// TIA Portal V17 export
// export: Created 2022-07-28T18:02:44.8373404Z, ExportSetting None, DisplayName Totally Integrated Automation Portal, DisplayVersion V17, DisplayName TIA Portal Openness, DisplayVersion V17, DisplayName TIA Portal Teamcenter Gateway, DisplayVersion V17, DisplayName TIA Portal Version Control Interface, DisplayVersion V17, DisplayName TIA Portal Test Suite Advanced, DisplayVersion V17, DisplayName SINAMICS Startdrive Advanced, DisplayVersion V17, DisplayName SINAMICS DCC, DisplayVersion V17, DisplayName SINAMICS Startdrive G130, G150, S120, S150, SINAMICS MV, S210, DisplayVersion V17, DisplayName SINAMICS Startdrive G110M, G120, G120C, G120D, G120P, G115D, DisplayVersion V17, DisplayName STEP 7 Professional, DisplayVersion V17, DisplayName SIMATIC Energy Suite, DisplayVersion V17, DisplayName STEP 7 CFC, DisplayVersion V17, DisplayName STEP 7 Safety, DisplayVersion V17, DisplayName WinCC Advanced / Unified PC, DisplayVersion V17, DisplayName SIMATIC Visualization Architect, DisplayVersion V17
FUNCTION_BLOCK "Lib_FB_PLC"   // FB1, SCL
{ S7_Optimized_Access := 'TRUE' }
// stored: MemoryReserve 500, SetENOAutomatically false
   VAR_IN_OUT
      IO_PLC : "Lib_UDT_PLC";
   END_VAR
   VAR
      TMBITS_PREV : Int;   // попереднє значення таймерних меандрів
      MEM_RUNTIME : LReal;   // память для вимірювання часу циклу
      FB_LTIME : LReal;
      FB_LTIME_1 : Real;
      TIME_TCK_ms : LReal;
      TIME_TCK_s : LReal;
      TIME_TCK_min : Real;
      TIME_TCK_ms_1 : DInt;
      TIME_TCK_ms_2 : UDInt;
      TIME_TCK_ms_3 : DInt;
      TIME_TCK_min_3rs : Real;
      OB1 : Struct
         PrevOutputTime : Date_And_Time;   // Время на предыдущего вызова
         cyclicTime : Int;   // Время цыкла (мс)
      END_STRUCT;
      TIME_ZONE : Struct
         Set : Bool;
         DONE : Bool;
         BUSY : Bool;
         ERROR : Bool;
         STATUS : Word;
         TimeTransformationRule : TimeTransformationRule;
      END_STRUCT;
      SET_TIMEZONE_Instance { ExternalAccessible := 'False'; ExternalVisible := 'False'; ExternalWritable := 'False'} : SET_TIMEZONE;
   END_VAR
   VAR_TEMP
      TMBITS_CUR : Int;
      RESULT : Int;
      i : Int;
      NOW : DTL;
      retVal : Int;
      test : LReal;
      TaskTimeMax : LTime;
      TaskTimeMin : LTime;
      TaskTimeLive : LTime;
      returnValue : Int;
   END_VAR
   // TIME_ZONE.TimeTransformationRule.Bias := 120;
   // TIME_ZONE.TimeTransformationRule.DaylightBias := 60;
   // TIME_ZONE.TimeTransformationRule.DaylightStartMonth := 3;
   // TIME_ZONE.TimeTransformationRule.DaylightStartWeek := 5;
   // TIME_ZONE.TimeTransformationRule.DaylightStartWeekday := 1;
   // TIME_ZONE.TimeTransformationRule.DaylightStartHour := 3;
   // TIME_ZONE.TimeTransformationRule.DaylightStartMinute := 0;
   // TIME_ZONE.TimeTransformationRule.StandardStartMonth := 10;
   // TIME_ZONE.TimeTransformationRule.StandardStartWeek := 5;
   // TIME_ZONE.TimeTransformationRule.StandardStartWeekday := 1;
   // TIME_ZONE.TimeTransformationRule.StandardStartHour := 3;
   // TIME_ZONE.TimeTransformationRule.StandardStartMinute := 0;
   // TIME_ZONE.TimeTransformationRule.TimeZoneName := '(GMT+02:00) Helsinki, Kiev, Riga, Sofia, Tallinn, Vilnius';
BEGIN
   //#FB_LTIME := RUNTIME(#MEM_RUNTIME) * 1000.0;



       REGION Iніціалізація "FirstScan"
           #IO_PLC.PLS.FirstScan := "FirstScan";
           IF #IO_PLC.PLS.FirstScan THEN (*при першому скані*)
               #IO_PLC.ID := 1;             (*Ідентифікатор завжди 1*)
               #IO_PLC.TIME_TCK.Time1cycle_r := 0;
               #TMBITS_CUR := 0;
               #TMBITS_PREV := 0;
           END_IF;
       END_REGION



   REGION таймерні біти та лічильники
       (*плинні значення*)
       REGION плинні значення
           #TMBITS_CUR.%X0 := "Clock_10Hz";         // 100MS 
           #TMBITS_CUR.%X1 := "Clock_5Hz";        // 200MS
           #TMBITS_CUR.%X2 := "Clock_2Hz";        // 500MS
           #TMBITS_CUR.%X3 := "Clock_1Hz";      // 1S
           #TMBITS_CUR.%X7 := #IO_PLC.NOW[0] > 16#29; //min
       END_REGION
       (*відловлювання імпульсів необхідних часових періодів*)
       REGION відловлювання імпульсів необхідних часових періодів
           #IO_PLC.PLS.P100MS := #TMBITS_CUR.%X0 AND NOT #TMBITS_PREV.%X0; (*100 мс *)
           #IO_PLC.PLS.P200MS := #TMBITS_CUR.%X1 AND NOT #TMBITS_PREV.%X1; (*200 мс*)
           #IO_PLC.PLS.P500MS := #TMBITS_CUR.%X2 AND NOT #TMBITS_PREV.%X2; (*500 мс*)
           #IO_PLC.PLS.P1S := #TMBITS_CUR.%X3 AND NOT #TMBITS_PREV.%X3; (*1 с*)
           #IO_PLC.PLS.P60S := #TMBITS_CUR.%X7 AND NOT #TMBITS_PREV.%X7; (*1 хв*)
       END_REGION
       (*підрахунок кількості секунд і хвилин*)
       (*загальний час з початку 1-го циклу контролера (в секундах)*)
       REGION загальний час з початку 1-го циклу контролера (в секундах)
           IF #IO_PLC.PLS.P1S THEN
               #IO_PLC.TIME_TCK.Time1cycle_di := #IO_PLC.TIME_TCK.Time1cycle_di + 1;
           END_IF;
           IF #IO_PLC.TIME_TCK.Time1cycle_di > 16#7FFF_FFFF THEN
               #IO_PLC.TIME_TCK.Time1cycle_di := 16#7FFF_FFFF;
           END_IF;
       END_REGION
       (*загальний час роботи ПЛК з моменту пуску (в хвилинах)*)
       REGION загальний час роботи ПЛК з моменту пуску (в хвилинах)
           IF #IO_PLC.PLS.P60S AND NOT #IO_PLC.PLS.FirstScan THEN
               #IO_PLC.TIME_TCK.TimeTotalPLC := #IO_PLC.TIME_TCK.TimeTotalPLC + 1;
           END_IF;
           IF #IO_PLC.TIME_TCK.TimeTotalPLC > 16#7FFF_FFFF THEN
               #IO_PLC.TIME_TCK.TimeTotalPLC := 16#7FFF_FFFF;
           END_IF;
       END_REGION
       (*розрахунок інших часових періодів*)
       REGION розрахунок інших часових періодів
           #IO_PLC.PLS.P2S := (#IO_PLC.TIME_TCK.Time1cycle_di MOD 2) = 0 AND #IO_PLC.PLS.P1S;(*2 с*)
           #IO_PLC.PLS.P5S := (#IO_PLC.TIME_TCK.Time1cycle_di MOD 5) = 0 AND #IO_PLC.PLS.P1S;(*5 с*)
           #IO_PLC.PLS.P10S := (#IO_PLC.TIME_TCK.Time1cycle_di MOD 10) = 0 AND #IO_PLC.PLS.P1S;(*10 с*)
           (* меандри *)
           #IO_PLC.PLS.M1S := "Clock_1Hz";  (*меандр з періодом 1 с (0.5 с + 0.5 с)*)
           #IO_PLC.PLS.M2S := "Clock_0.5Hz";(*меандр з періодом 2 с (1 с + 1 с) *)
           (* початок години *)
           #IO_PLC.PLS.NEWHR := (#IO_PLC.NOW[1] AND 16#00FF) = 0 (*хвилини*)AND #IO_PLC.PLS.P60S (*один раз за хвилину*);
           (* початок доби*)
           #IO_PLC.PLS.NEWDAY := #IO_PLC.NOW[1] = 0 (*години_хвилини*)AND #IO_PLC.PLS.P60S (*один раз за хвилину*);
       END_REGION
       #TMBITS_PREV := #TMBITS_CUR;(*збереження попередніх значень*)
   END_REGION

   REGION астрономічний час
       REGION Поточний час
           (*+*) #RESULT := RD_LOC_T(#NOW);
           (*+*) #IO_PLC.TIME_TCK.NowTime := #NOW;
           #IO_PLC.NOW[0] :=INT_TO_BCD16(#NOW.SECOND); //#NOW[0] seconds,-- (16#ss,--)
           #IO_PLC.NOW[1] := SHL(IN := INT_TO_BCD16(#NOW.HOUR), N := 8) OR INT_TO_BCD16(#NOW.MINUTE);//16#hhmm
           #IO_PLC.NOW[2] := SHL(IN := INT_TO_BCD16(#NOW.MONTH), N := 8) OR INT_TO_BCD16(#NOW.DAY);  //16#mmdd
           #IO_PLC.NOW[3] := SHL(IN := INT_TO_BCD16(#NOW.YEAR / 100), N := 8) OR INT_TO_BCD16(#NOW.YEAR MOD 100);
       END_REGION
       REGION Встановити годину

       END_REGION
   END_REGION

   REGION Зміни
       (*початок зміни*)
       REGION початок зміни
           IF #IO_PLC.ShiftParam[0] < 1 OR #IO_PLC.ShiftParam[0] > 3 THEN
               #IO_PLC.ShiftParam[0] := 2;
           END_IF;(*коректність кількості змін*)
           #IO_PLC.PLS.NEWSHIFT := FALSE; (*скидуємо біт початку зміни*)
           FOR #i := 1 TO #IO_PLC.ShiftParam[0] DO
               (*хоча б одна з устоавок змін спрацювала*)
               #IO_PLC.PLS.NEWSHIFT := #IO_PLC.PLS.NEWSHIFT OR (#IO_PLC.ShiftParam[#i] = #IO_PLC.NOW[1] (*години хвилин*)AND #IO_PLC.PLS.P60S (*один раз за хвилину*));
           END_FOR;
       END_REGION
       // (*----------- визначеня зміни*)
       REGION визначеня зміни
           IF #IO_PLC.ShiftParam[0] > 3 OR #IO_PLC.ShiftParam[0] < 2 THEN
               #IO_PLC.ShiftParam[0] := 3;
           END_IF;(*якщо кількість змін >3 або <1 - робимо 3*)
           IF #IO_PLC.NOW[1] >= #IO_PLC.ShiftParam[1] AND (#IO_PLC.NOW[1] < #IO_PLC.ShiftParam[2] OR #IO_PLC.ShiftParam[2] = 16#0000) THEN (*1-ша зміна*)
               #IO_PLC.ShiftActiveNumber := 1;
           ELSE (*2-га або 3-тя*)
               IF #IO_PLC.ShiftParam[0] = 2 THEN (*якщо в 2 зміни*)
                   #IO_PLC.ShiftActiveNumber := 2;
               ELSE (*якщо 3 зміни*)
                   IF #IO_PLC.NOW[1] >= #IO_PLC.ShiftParam[2] AND (#IO_PLC.NOW[1] < #IO_PLC.ShiftParam[3] OR #IO_PLC.ShiftParam[3] = 16#0000) THEN
                       #IO_PLC.ShiftActiveNumber := 2;
                   ELSE
                       #IO_PLC.ShiftActiveNumber := 3;
                   END_IF;
               END_IF;
           END_IF;
       END_REGION

   END_REGION
   //#FB_LTIME := RUNTIME(#MEM_RUNTIME) * 1000.0;

   // #test := 2;
   // FOR #i := 1 TO 100 DO
   //     (*хоча б одна з устоавок змін спрацювала*)
   //     #test := #test ** #i;
   // END_FOR;
   //#FB_LTIME := RUNTIME(#MEM_RUNTIME) * 1000.0;


   //
   REGION Час циклу

       IF NOT "FirstScan" THEN
          (*+for cyclic_sec_R*) #IO_PLC.TIME_TCK.cyclic_ms := TIME_TO_INT(#IO_PLC.TIME_TCK.NowTime - #IO_PLC.TIME_TCK.PrevScanTime);
          (*+for cyclic_sec_R*) #IO_PLC.TIME_TCK.PrevScanTime := #IO_PLC.TIME_TCK.NowTime;
          (*+for cyclic_sec_R*) #IO_PLC.TIME_TCK.cyclic_sec_LR := INT_TO_LREAL(#IO_PLC.TIME_TCK.cyclic_ms) / 1000;
          (*+for cyclic_sec_R*) #IO_PLC.TIME_TCK.cyclic_sec_R := LREAL_TO_REAL(#IO_PLC.TIME_TCK.cyclic_sec_LR);
           #IO_PLC.TIME_TCK.Time1cycle_r := #IO_PLC.TIME_TCK.Time1cycle_r + #IO_PLC.TIME_TCK.cyclic_sec_LR;//TIME_TO_LINT(#IO_PLC.TIME_TCK.NowTime - #IO_PLC.TIME_TCK.FirstScanTime)/1000;
           #IO_PLC.TIME_TCK.Time1cycle_DINT := LREAL_TO_UDINT(#IO_PLC.TIME_TCK.Time1cycle_r);

       ELSE
           #IO_PLC.TIME_TCK.FirstScanTime := #IO_PLC.TIME_TCK.NowTime;
           #IO_PLC.TIME_TCK.PrevScanTime := #IO_PLC.TIME_TCK.NowTime;
           #IO_PLC.TIME_TCK.Time1cycle_r := 0;
           #IO_PLC.TIME_TCK.Time1cycle_DINT := 0;

       END_IF;
   END_REGION





   REGION Час циклу PLC з RT_INFO
       IF NOT "FirstScan" THEN
           #FB_LTIME := RUNTIME(#MEM_RUNTIME);
           #FB_LTIME_1 := LREAL_TO_REAL(#FB_LTIME);
           //#TIME_TCK_ms := #TIME_TCK_ms + #FB_LTIME;
           #TIME_TCK_s := #TIME_TCK_s + #FB_LTIME;//LREAL_TO_REAL(#TIME_TCK_ms/1000);
           #TIME_TCK_min := #TIME_TCK_s;

           //#TIME_TCK_ms_3 := #TIME_TCK_ms_3 + #OB1.cyclicTime;
           //#TIME_TCK_min_3rs := DINT_TO_REAL(#TIME_TCK_ms_3) / 1000;
           IF #IO_PLC.PLS.P100MS THEN
               #TIME_TCK_ms_1 := #TIME_TCK_ms_1 + 100;
               #TIME_TCK_ms_2 := LREAL_TO_DINT(#TIME_TCK_s * 1000);
           END_IF;
       ELSE
           #TIME_TCK_s := 0;
           #MEM_RUNTIME := 0;
           #TIME_TCK_ms_1 := 0;
           #TIME_TCK_ms_1 := 0;
           #TIME_TCK_ms_3 := 0;
           #IO_PLC.TaskTime_RUNTIME.TIME_TCK_s := 0;

       END_IF;
   END_REGION


   REGION Час циклу PLC з RT_INFO
   (*цикли*)
       //!!!!s7-1200 not suport RT_INFO
   //#PLC.TSK_LTIME_1 := LREAL_TO_UINT(RUNTI1ME(#MEM_RT) * 1000.0);
   //#retVal := RT_INFO(MODE := 23, OB := 1, INFO := #TaskTimeMax);
   //#retVal := RT_INFO(MODE := 24, OB := 1, INFO := #TaskTimeMin);
   //#retVal := RT_INFO(MODE := 25, OB := 1, INFO := #TaskTimeLive);
   //#IO_PLC.TaskTime.Max := ULINT_TO_LREAL(LTIME_TO_ULINT(#TaskTimeMax)) / 1000000;
   //#IO_PLC.TaskTime.Min := ULINT_TO_LREAL(LTIME_TO_ULINT(#TaskTimeMin)) / 1000000;
   //#IO_PLC.TaskTime.Live := ULINT_TO_LREAL(LTIME_TO_ULINT(#TaskTimeLive)) / 1000000;
   //#IO_PLC.TaskTime_RUNTIME.Live := #IO_PLC.TaskTime.Live;
   //#IO_PLC.TaskTime_RUNTIME.TIME_TCK_s := (#IO_PLC.TaskTime_RUNTIME.TIME_TCK_s + #IO_PLC.TaskTime_RUNTIME.Live / 1000);

   //!!!!!!!
   #TIME_TCK_ms := #IO_PLC.TaskTime_RUNTIME.TIME_TCK_s;

   END_REGION
   REGION sET TIME ZONE
       // Statement section REGION
       #SET_TIMEZONE_Instance(REQ := #TIME_ZONE.Set,
                              TimeZone := #TIME_ZONE.TimeTransformationRule,
                              DONE => #TIME_ZONE.DONE,
                              BUSY => #TIME_ZONE.BUSY,
                              ERROR => #TIME_ZONE.ERROR,
                              STATUS => #TIME_ZONE.STATUS);
   END_REGION
END_FUNCTION_BLOCK
